Fanuc KAREL source: CURR_PROG.kl

PROGRAM T
%NOLOCKGROUP
VAR
 res : STRING[40]
BEGIN
 res = CURR_PROG
END T
